(* PLC project , Beckhoff Automation GmbH TwinCAT PLC Control 3.5.13.21 *)
(* stored: creationDateTime 2025-04-03T13:53:02.3507151 *)

{attribute 'qualified_only'}
{attribute 'strict'}
TYPE E_State :
(
	None,
	Init,
	StartingMotor,
	OpeningFile,
	Chirp,
	Saving,
	SlowingDown,
	Stopping,
	DisableMotor
);
END_TYPE
